TYPE TFMachinePalletizer_OUT :
STRUCT
	Run : BOOL;
	Warning : BOOL;
	Error : BOOL;
	Horn : BOOL;
	StartHorn : BOOL;

	PowerActive : BOOL;
	
	HomeDone : BOOL;
	
	StopTilterReq : BOOL;
	PowerOffTilterReq : BOOL;
	PowerOnTilterReq : BOOL;
	ResetTilterReq : BOOL;
	StartTilter : BOOL;
	
	ClockSegnalazioni : bool;//Clock per segnalazioni varie
	
	PowerActiveSIMULAZIONE : BOOL;
	
	ClockSegnalazioniAlternato	: BOOL;//Clock Segnalazioni  Alternato
	ResetSirenaSegnalazioni : BOOL; //Segnale di stop suoneria sirena 
END_STRUCT
END_TYPE

(* stored: Version 1.1.0.1, ProductVersion 3.1.4024.11
   DUT TFMachinePalletizer_OUT: Id {ebfdbb7b-cc54-4a8a-8fc8-6e5ef102a781} *)
